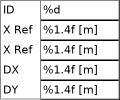
VISUALIZATION _VISU_DeformationPoint  // 120x100
VAR_IN_OUT
	m_Inst : ST_DeformationPointAccurate;
END_VAR
    Rectangle (40,0 80x20), "%d", text variable: m_Inst.index
    Rectangle (0,0 40x20), "ID"
    Rectangle (40,20 80x20), "%1.4f [m]", text variable: m_Inst.x_ref
    Rectangle (0,20 40x20), "X Ref"
    Rectangle (40,40 80x20), "%1.4f [m]", text variable: m_Inst.y_ref
    Rectangle (0,40 40x20), "X Ref"
    Rectangle (40,60 80x20), "%1.4f [m]", text variable: m_Inst.dx
    Rectangle (0,60 40x20), "DX"
    Rectangle (40,80 80x20), "%1.4f [m]", text variable: m_Inst.dy
    Rectangle (0,80 40x20), "DY"
END_VISUALIZATION

(* stored: Version 1.1.0.1, ProductVersion 3.1.4024.3
   Visu _VISU_DeformationPoint: Id {b49a5385-0c28-4714-b082-b343785afafb} *)
